Staubli VAL3: start.pgx

program start()
begin

  // Blank interface library to load at runtime
  // The correct library will be loaded in the application

end
